(* IEC 61131-3 sources: ST_DesignPattern/Behavioral, 4 files *)

(* ---- adapter.st ---- *)
{attribute 'qualified_only'}
{attribute 'strict'}
{attribute 'to_string'}
TYPE E_GasSystemType:
(
    PRECURSOR := 0,
    REACTANT := 1,
    INERT := 2
);
END_TYPE

{attribute 'qualified_only'}
{attribute 'strict'}
{attribute 'to_string'}
TYPE E_MFCState:
(
    Idle := 0,
    Running := 10,
    Error := 20
);
END_TYPE

TYPE ST_MFCConfig :
STRUCT
    fMaxFlow    : REAL;
    fMinFlow    : REAL;
    fTolerance  : REAL;
    sName       : STRING;
    sFlowUnit   : STRING := 'sccm';
END_STRUCT
END_TYPE

INTERFACE I_MFC
    METHOD SetFlow : BOOL
    VAR_INPUT
        fSetpoint : REAL;
    END_VAR
    END_METHOD

    METHOD GetFlow : REAL
    END_METHOD

    METHOD AtSetpoint : BOOL
    END_METHOD

    METHOD Stop : BOOL
    END_METHOD

    PROPERTY State : E_MFCState GET
    END_PROPERTY

    PROPERTY Error : ST_Error GET
    END_PROPERTY
END_INTERFACE

FUNCTION_BLOCK FB_MFC IMPLEMENTS I_MFC
VAR
    _config : ST_MFCConfig;
    _state : E_MFCState := E_MFCState.Idle;
    _errorHandler : FB_ErrorHandler;
    _pMFC : POINTER TO massFlowController;
END_VAR

VAR CONSTANT
    ZERO_FLOW_THRESHOLD : REAL := 0.001;
END_VAR

METHOD Initialize : BOOL
VAR_INPUT
    config: ST_MFCConfig;
    pMFC: POINTER TO massFlowController;
END_VAR
    _config := config;
    _pMFC := pMFC;
    _errorHandler := errorHandler;

    IF _pMFC = 0 THEN
        _errorHandler.RegisterError(
            eErrorCode := E_ErrorCodes.NotInitialized,
            eCategory := E_ErrorCategory.Hardware,
            sComponent := _config.sName,
            sDescription := 'MFC hardware not connected',
            sCurrentValue := '',
            sExpectedValue := '',
            sUnit := ''
        );
        _state := E_MFCState.Error;
        Initialize := FALSE;
        RETURN;
    END_IF

    Initialize := TRUE;
END_METHOD

METHOD SetFlow : BOOL
VAR_INPUT
    fSetpoint : REAL;
END_VAR
    IF _pMFC = 0 THEN
        _errorHandler.RegisterError(
            eErrorCode := E_ErrorCodes.NotInitialized,
            eCategory := E_ErrorCategory.Hardware,
            sComponent := _config.sName,
            sDescription := 'MFC hardware not connected',
            sCurrentValue := '',
            sExpectedValue := '',
            sUnit := ''
        );
        _state := E_MFCState.Error;
        SetFlow := FALSE;
        RETURN;
    END_IF

    IF fSetpoint < _config.fMinFlow OR fSetpoint > _config.fMaxFlow THEN
        _errorHandler.RegisterError(
            eErrorCode := E_ErrorCodes.FlowOutOfRange,
            eCategory := E_ErrorCategory.FlowControl,
            sComponent := _config.sName,
            sDescription := 'Flow setpoint out of range',
            sCurrentValue := REAL_TO_STRING(fSetpoint),
            sExpectedValue := CONCAT(LREAL_TO_STRING(_config.fMinFlow), CONCAT(' - ', LREAL_TO_STRING(_config.fMaxFlow))),
            sUnit := 'sccm'
        );
        _state := E_MFCState.Error;
        RETURN;
    END_IF

    _pMFC^.SetPointIn := fSetpoint;
    _state := SEL(fSetpoint = 0, E_MFCState.Running, E_MFCState.Idle);
    SetFlow := TRUE;
END_METHOD

METHOD GetFlow : REAL
    IF _pMFC <> 0 THEN
        GetFlow := _pMFC^.ProcessValue;
    END_IF
END_METHOD

METHOD AtSetpoint : BOOL
    IF _pMFC = 0 THEN
        AtSetpoint := FALSE;
        RETURN;
    END_IF

    AtSetpoint := ABS(_pMFC^.ProcessValue - _pMFC^.SetPointIn) <= (_pMFC^.SetPointIn * _config.fTolerance / 100.0);
END_METHOD

METHOD Stop : BOOL
    Stop := SetFlow(0.0);
END_METHOD

PROPERTY State : E_MFCState GET
    State := _state;
END_PROPERTY

PROPERTY Error : ST_Error GET
    Error := _errorHandler.GetError();
END_PROPERTY
END_FUNCTION_BLOCK

FUNCTION_BLOCK FB_DualMFC IMPLEMENTS I_MFC
VAR
    _highFlow: FB_MFC;
    _lowFlow: FB_MFC;
    _flowThreshold: REAL;
    _activeFlow: REFERENCE TO FB_MFC;
    _state: E_MFCState := E_MFCState.Idle;
    _errorHandler: FB_ErrorHandler;
END_VAR

METHOD Initialize : BOOL
VAR_INPUT
    highConfig: ST_MFCConfig;
    lowConfig: ST_MFCConfig;
    pHighMFC: POINTER TO massFlowController;
    pLowMFC: POINTER TO massFlowController;
    errorHandler: I_ErrorHandler;
END_VAR
    _errorHandler := errorHandler;

    IF NOT _highFlow.Initialize(highConfig, pHighMFC, _errorHandler) THEN
        _errorHandler.RegisterError(
            eErrorCode := E_ErrorCodes.MFCTimeout,
            eCategory := E_ErrorCategory.Initialization,
            sComponent := 'DualMFC-High',
            sDescription := 'Failed to initialize high flow MFC',
            sCurrentValue := '',
            sExpectedValue := '',
            sUnit := ''
        );
        _state := E_MFCState.Error;
        RETURN FALSE;
    END_IF

    IF NOT _lowFlow.Initialize(lowConfig, pLowMFC, _errorHandler) THEN
        _errorHandler.RegisterError(
            eErrorCode := E_ErrorCodes.MFCTimeout,
            eCategory := E_ErrorCategory.Initialization,
            sComponent := 'DualMFC-Low',
            sDescription := 'Failed to initialize low flow MFC',
            sCurrentValue := '',
            sExpectedValue := '',
            sUnit := ''
        );
        _state := E_MFCState.Error;
        RETURN FALSE;
    END_IF

    _flowThreshold := lowConfig.fMaxFlow;
    _activeFlow REF= _lowFlow;
    _state := E_MFCState.Idle;
    Initialize := TRUE;
END_METHOD

METHOD SetFlow : BOOL
VAR_INPUT
    fSetpoint : REAL;
END_VAR
    IF _state = E_MFCState.Error THEN
        RETURN FALSE;
    END_IF

    IF fSetpoint <= _flowThreshold THEN
        _highFlow.Stop();
        _activeFlow REF= _lowFlow;
    ELSE
        _lowFlow.Stop();
        _activeFlow REF= _highFlow;
    END_IF

    SetFlow := _activeFlow.SetFlow(fSetpoint);
    _state := _activeFlow.State;
END_METHOD

METHOD GetFlow : REAL
    GetFlow := _lowFlow.GetFlow() + _highFlow.GetFlow();
END_METHOD

METHOD Stop : BOOL
    _highFlow.Stop();
    _lowFlow.Stop();
    _state := E_MFCState.Idle;
    Stop := TRUE;
END_METHOD

METHOD AtSetpoint : BOOL
    IF _state = E_MFCState.Error THEN
        RETURN FALSE;
    END_IF

    AtSetpoint := _activeFlow.AtSetpoint();
END_METHOD

PROPERTY State : E_MFCState GET
    State := _state;
END_PROPERTY

PROPERTY Error : ST_Error GET
    IF _activeFlow.State = E_MFCState.Error THEN
        Error := _activeFlow.Error;
    ELSE
        Error := _errorHandler.GetError();
    END_IF
END_PROPERTY
END_FUNCTION_BLOCK

FUNCTION_BLOCK FB_MFCFactory
VAR CONSTANT
    PRECURSOR_HIGH_CONFIG : ST_MFCConfig := (
        fMaxFlow := 2000.0,
        fMinFlow := 400.0,
        fTolerance := 2.0,
        sName := 'Precursor High Flow',
        sFlowUnit := 'sccm'
    );

    PRECURSOR_LOW_CONFIG : ST_MFCConfig := (
        fMaxFlow := 400.0,
        fMinFlow := 0.0,
        fTolerance := 2.0,
        sName := 'Precursor Low Flow',
        sFlowUnit := 'sccm'
    );

    REACTANT_CONFIG : ST_MFCConfig := (
        fMaxFlow := 1000.0,
        fMinFlow := 0.0,
        fTolerance := 2.0,
        sName := 'Reactant Flow',
        sFlowUnit := 'sccm'
    );

    INERT_HIGH_CONFIG : ST_MFCConfig := (
        fMaxFlow := 5000.0,
        fMinFlow := 400.0,
        fTolerance := 2.0,
        sName := 'Inert High Flow',
        sFlowUnit := 'sccm'
    );

    INERT_LOW_CONFIG : ST_MFCConfig := (
        fMaxFlow := 400.0,
        fMinFlow := 0.0,
        fTolerance := 2.0,
        sName := 'Inert Low Flow',
        sFlowUnit := 'sccm'
    );
END_VAR

VAR
    _reactantMFC : FB_MFC;
    _precursorDualMFC : FB_DualMFC;
    _inertDualMFC : FB_DualMFC;
    _errorHandler : I_ErrorHandler;
    _bInitialized : BOOL := FALSE;

END_VAR

METHOD Initialize : BOOL
VAR_INPUT
    bResetError : BOOL := FALSE;
    errorHandler : I_ErrorHandler;
END_VAR
    _errorHandler := errorHandler;

    IF bResetError THEN
        _errorHandler.Reset();
    END_IF

    IF _bInitialized THEN
        Initialize := TRUE;
        RETURN;
    END_IF

    IF NOT _reactantMFC.Initialize(REACTANT_CONFIG, ADR(GVL_E02_MFC.MFC.st_MFC.ReactantMassFlowController1), _errorHandler) THEN
        _errorHandler.RegisterError(
            eErrorCode := E_ErrorCodes.MFCTimeout,
            eCategory := E_ErrorCategory.Initialization,
            sComponent := REACTANT_CONFIG.sName,
            sDescription := 'Failed to initialize reactant MFC',
            sCurrentValue := '',
            sExpectedValue := '',
            sUnit := REACTANT_CONFIG.sFlowUnit
        );
        RETURN;
    END_IF

    IF NOT _precursorDualMFC.Initialize(PRECURSOR_HIGH_CONFIG, PRECURSOR_LOW_CONFIG, ADR(GVL_E02_MFC.MFC.st_MFC.PrecursorMassFlowController1), ADR(GVL_E02_MFC.MFC.st_MFC.PrecursorMassFlowController2), _errorHandler) THEN
        _errorHandler.RegisterError(
            eErrorCode := E_ErrorCodes.MFCTimeout,
            eCategory := E_ErrorCategory.Initialization,
            sComponent := 'Precursor Dual MFC',
            sDescription := 'Failed to initialize precursor dual MFC',
            sCurrentValue := '',
            sExpectedValue := '',
            sUnit := PRECURSOR_HIGH_CONFIG.sFlowUnit
        );
        RETURN;
    END_IF

    IF NOT _inertDualMFC.Initialize(INERT_HIGH_CONFIG, INERT_LOW_CONFIG, ADR(GVL_E02_MFC.MFC.st_MFC.InertMassFlowController1), ADR(GVL_E02_MFC.MFC.st_MFC.InertMassFlowController2), _errorHandler) THEN
        _errorHandler.RegisterError(
            eErrorCode := E_ErrorCodes.MFCTimeout,
            eCategory := E_ErrorCategory.Initialization,
            sComponent := 'Inert Dual MFC',
            sDescription := 'Failed to initialize inert dual MFC',
            sCurrentValue := '',
            sExpectedValue := '',
            sUnit := INERT_HIGH_CONFIG.sFlowUnit
        );
        RETURN;
    END_IF

    _bInitialized := TRUE;
    Initialize := TRUE;
END_METHOD

METHOD GetController : REFERENCE TO I_MFC
VAR_INPUT
    eGasType : E_GasSystemType;
END_VAR
    IF NOT _bInitialized THEN
        _errorHandler.RegisterError(
            eErrorCode := E_ErrorCodes.NotInitialized,
            eCategory := E_ErrorCategory.Initialization,
            sComponent := 'MFCFactory',
            sDescription := 'Factory not initialized',
            sCurrentValue := '',
            sExpectedValue := '',
            sUnit := ''
        );
        RETURN;
    END_IF

    CASE eGasType OF
        E_GasSystemType.PRECURSOR:
            GetController REF= _precursorDualMFC;

        E_GasSystemType.REACTANT:
            GetController REF= _reactantMFC;

        E_GasSystemType.INERT:
            GetController REF= _inertDualMFC;

        ELSE
            _errorHandler.RegisterError(
                eErrorCode := E_ErrorCodes.InvalidConfiguration,
                eCategory := E_ErrorCategory.FlowControl,
                sComponent := 'MFCFactory',
                sDescription := 'Invalid gas system type',
                sCurrentValue := TO_STRING(eGasType),
                sExpectedValue := 'PRECURSOR, REACTANT, or INERT',
                sUnit := ''
            );
    END_CASE
END_METHOD

PROPERTY Error : ST_Error GET
    Error := _errorHandler.GetError();
END_PROPERTY
END_FUNCTION_BLOCK

(* ---- bridge.st ---- *)
FUNCTION_BLOCK ABSTRACT FB_Shape
VAR
	_color : ITF_color;
END_VAR
    METHOD FB_init : BOOL
    VAR_INPUT
        bInitRetains : BOOL; // if TRUE, the retain variables are initialized (warm start / cold start)
        bInCopyCode : BOOL;  // if TRUE, the instance afterwards gets moved into the copy code (online change)
        Color : ITF_Color;
    END_VAR
        THIS^._color := Color;
    END_METHOD

    METHOD ABSTRACT Draw : STRING
    END_METHOD
END_FUNCTION_BLOCK

FUNCTION_BLOCK FB_Square EXTENDS FB_Shape
    METHOD Draw : STRING
        ADSLOGSTR(    msgCtrlMask:=ADSLOG_MSGTYPE_LOG,
              msgFmtStr:='Drawing a %s square',
              strArg:= SUPER^._color.applyColor());
    END_METHOD
END_FUNCTION_BLOCK

FUNCTION_BLOCK FB_Circle EXTENDS FB_Shape
    METHOD Draw : STRING
        ADSLOGSTR(    msgCtrlMask:=ADSLOG_MSGTYPE_LOG,
              msgFmtStr:='Drawing a %s circle',
              strArg:= SUPER^._color.applyColor());
    END_METHOD
END_FUNCTION_BLOCK

INTERFACE ITF_Color
    METHOD applyColor : STRING
    END_METHOD
END_INTERFACE

FUNCTION_BLOCK FB_BlueColor IMPLEMENTS ITF_Color
    METHOD applyColor : STRING
        applyColor := 'blue';
    END_METHOD
END_FUNCTION_BLOCK

FUNCTION_BLOCK FB_RedColor IMPLEMENTS ITF_Color
    METHOD applyColor : STRING
        applyColor := 'red';
    END_METHOD
END_FUNCTION_BLOCK

PROGRAM MAIN
VAR

     fbRedColor 		: FB_RedColor;
	 fbBlueColor 		: FB_BlueColor;

	 fbSquareRed 		: FB_Square(Color:= fbRedColor );
	 fbSquareBlue 		: FB_Square(Color:= fbBlueColor );

	 fbCircleRed 		: FB_Circle(Color:= fbRedColor );
	 fbCircleBlue 		: FB_Circle(Color:= fbBlueColor );

	 bstartDemo1		: BOOL;

END_VAR
    IF bstartDemo1 THEN
        bstartDemo1 := FALSE;

        fbSquareRed.Draw();
        fbSquareBlue.Draw();

        fbCircleRed.Draw();
        fbCircleBlue.Draw();

    END_IF
END_PROGRAM

(* ---- composite.st ---- *)
INTERFACE I_Component
    METHOD AddChild
    VAR_INPUT
        Child : I_Component;
    END_VAR
    END_METHOD

    METHOD GetChildren : ARRAY [1..Param.NumberOfChildren] OF I_Component;
    END_METHOD

    PROPERTY GetSize : INT GET
    END_PROPERTY
END_INTERFACE

FUNCTION_BLOCK ABSTRACT Component IMPLEMENTS I_component
VAR
	_name : STRING;
END_VAR
    METHOD FB_init : BOOL
    VAR_INPUT
        bInitRetains : BOOL; // if TRUE, the retain variables are initialized (warm start / cold start)
        bInCopyCode : BOOL;  // if TRUE, the instance afterwards gets moved into the copy code (online change)
        name : STRING;
    END_VAR
    THIS^._name := name;
    END_METHOD

    METHOD ABSTRACT AddChild
    VAR_INPUT
        Child : I_Component;
    END_VAR
    END_METHOD

    METHOD ABSTRACT GetChildren : ARRAY [1..Param.NumberOfChildren] OF I_Component;
    END_METHOD

    PROPERTY ABSTRACT GetSize : INT GET
    END_PROPERTY

    PROPERTY Name : STRING GET
        Name := THIS^._name;
    END_PROPERTY
END_FUNCTION_BLOCK

FUNCTION_BLOCK Archive EXTENDS Component
VAR
//	_name : STRING;
	_size : INT;
END_VAR
    METHOD FB_init : BOOL
    VAR_INPUT
        bInitRetains : BOOL; // if TRUE, the retain variables are initialized (warm start / cold start)
        bInCopyCode : BOOL;  // if TRUE, the instance afterwards gets moved into the copy code (online change)
        name : STRING;
        iSize : INT;
    END_VAR
        THIS^._name := name;
        THIS^._size := iSize
    END_METHOD

    METHOD AddChild
    VAR_INPUT
        Child : I_Component;
    END_VAR
    END_METHOD

    METHOD GetChildren : ARRAY [1..Param.NumberOfChildren] OF I_Component;
    VAR_INPUT
    END_VAR
    END_METHOD

    PROPERTY GetSize : INT GET
        GetSize := _size;
    END_PROPERTY
END_FUNCTION_BLOCK

FUNCTION_BLOCK Directory EXTENDS Component
VAR
	children 			: ARRAY [1..Param.NumberOfChildren] OF I_Component;
	childCount			: INT := 0;
END_VAR
    METHOD AddChild
    VAR_INPUT
        Child : I_Component;
    END_VAR
    VAR
        i: INT;
    END_VAR
        childCount := childCount + 1;
        children[childCount] := Child;
    END_METHOD

    METHOD GetChildren : ARRAY [1..Param.NumberOfChildren] OF I_Component;
        GetChildren := children;
    END_METHOD

    PROPERTY GetSize : INT
    VAR
        i : INT := 0;
    END_VAR
        FOR i := 1 TO childCount  DO
            GetSize := GetSize + children[i].GetSize;
        END_FOR
    END_PROPERTY

    METHOD ResetSize
        childCount:= 0;
    END_METHOD
END_FUNCTION_BLOCK

PROGRAM MAIN
VAR
	root 		: Directory('root');

	archive1	: Archive('archivo1.txt', 10);
    archive2  	: Archive('archivo2.txt', 30);
    archive3 	: Archive('archivo3.txt', 120);
    archive4 	: Archive('archivo4.txt', 800);
    archive5 	: Archive('archivo5.txt', 340);

    archive6 	: Archive('archivo6.txt', 122);
    archive7 	: Archive('archivo7.txt', 391);

    dir1 		: Directory('dir1');
    dir2 		: Directory('dir2');
    dir3 		: Directory('dir3');

	bExecute	: BOOL;
	sMsg 		: STRING;
END_VAR
    IF bExecute THEN

        bExecute := FALSE;

        dir1.ResetSize();
        dir2.ResetSize();
        dir3.ResetSize();
        root.ResetSize();

        dir1.AddChild(archive1); // 10
        dir1.AddChild(archive6); // 122
        dir2.AddChild(archive2); // 30
        dir3.AddChild(archive3); // 120
        dir3.AddChild(archive4); // 800
        dir1.AddChild(dir3); // 120+800

        root.AddChild(dir1); // dir1 = 120+800+10+122 = 1052
        root.AddChild(dir2); // dir2 = 30
        root.AddChild(archive5); // 340
        root.AddChild(archive7); // 391

        // root = 1052+30+340+391 = 1813
        sMsg := CONCAT(STR1:= root.Name , STR2:= CONCAT(STR1:= ' is: ' , STR2:= TO_STRING(root.GetSize) ) );
        ADSLOGSTR(msgCtrlMask:= ADSLOG_MSGTYPE_LOG, msgFmtStr:= 'The size of the directory %s ' , strArg:= sMsg);

        // dir1 = 10+122+120+800 = 1052
        sMsg := CONCAT(STR1:= dir1.Name , STR2:= CONCAT(STR1:= ' is: ' , STR2:= TO_STRING(dir1.GetSize) ) );
        ADSLOGSTR(msgCtrlMask:= ADSLOG_MSGTYPE_LOG, msgFmtStr:= 'The size of the directory %s ' , strArg:= sMsg);

        // dir2 = 30
        sMsg := CONCAT(STR1:= dir2.Name , STR2:= CONCAT(STR1:= ' is: ' , STR2:= TO_STRING(dir2.GetSize) ) );
        ADSLOGSTR(msgCtrlMask:= ADSLOG_MSGTYPE_LOG, msgFmtStr:= 'The size of the directory %s ' , strArg:= sMsg);

        // dir3 = 120+800 = 922
        sMsg := CONCAT(STR1:= dir3.Name , STR2:= CONCAT(STR1:= ' is: ' , STR2:= TO_STRING(dir3.GetSize) ) );
        ADSLOGSTR(msgCtrlMask:= ADSLOG_MSGTYPE_LOG, msgFmtStr:= 'The size of the directory %s ' , strArg:= sMsg);
    END_IF
END_PROGRAM

(* ---- decorator.st ---- *)
INTERFACE I_Shape
    METHOD M_Draw: BOOL
    END_METHOD
END_INTERFACE

FUNCTION_BLOCK FB_Circle IMPLEMENTS I_Shape
    METHOD M_Draw: BOOL
        ADSLOGSTR(ADSLOG_MSGTYPE_HINT, 'Draw circle', '');
        M_Draw := TRUE;
    END_METHOD
END_FUNCTION_BLOCK

FUNCTION_BLOCK FB_Square IMPLEMENTS I_Shape
    METHOD M_Draw: BOOL
        ADSLOGSTR(ADSLOG_MSGTYPE_HINT, 'Draw Square', '');
        M_Draw := TRUE;
    END_METHOD
END_FUNCTION_BLOCK

FUNCTION_BLOCK ABSTRACT FB_ShapeDecorator IMPLEMENTS I_Shape
VAR
	_iDecoratedShape: I_Shape;
END_VAR
    METHOD FB_init: BOOL
    VAR_INPUT
        bInitRetains: BOOL; // if TRUE, the retain variables are initialized (warm start / cold start)
        bInCopyCode: BOOL; // if TRUE, the instance afterwards gets moved into the copy code (online change)
        iDecoratedShape: I_Shape;
    END_VAR
        _iDecoratedShape := iDecoratedShape;
    END_METHOD

    METHOD ABSTRACT M_Draw: BOOL
    END_METHOD
END_FUNCTION_BLOCK

{attribute 'qualified_only'}
{attribute 'strict'}
TYPE E_BorderDashType:
(
	Solid := 0,
	RoundDot,
	SquareDot,
	Dash,
	LongDashDot
);
END_TYPE

FUNCTION_BLOCK FB_BorderDashTypeDecorator EXTENDS FB_ShapeDecorator
VAR
	_eBorderDashType: E_BorderDashType;
END_VAR
    METHOD FB_init: BOOL
    VAR_INPUT
        bInitRetains: BOOL; // if TRUE, the retain variables are initialized (warm start / cold start)
        bInCopyCode: BOOL; // if TRUE, the instance afterwards gets moved into the copy code (online change)
        iDecoratedShape: I_Shape;
        eBorderDashType: E_BorderDashType;
    END_VAR
        SUPER^._iDecoratedShape := iDecoratedShape;
        _eBorderDashType := eBorderDashType;
    END_METHOD

    METHOD M_Draw: BOOL
        M_Draw := SUPER^._iDecoratedShape.M_Draw();
        M_SetBorderDashType(SUPER^._iDecoratedShape);
    END_METHOD

    METHOD M_SetBorderDashType
    VAR_INPUT
        iDecoratedShape: I_Shape;
    END_VAR
        CASE _eBorderDashType OF
            E_BorderDashType.Solid:
                ADSLOGSTR(ADSLOG_MSGTYPE_HINT, 'Border Dash Type: Solid', '');

            E_BorderDashType.SquareDot:
                ADSLOGSTR(ADSLOG_MSGTYPE_HINT, 'Border Dash Type: Square Dot', '');

            E_BorderDashType.RoundDot:
                ADSLOGSTR(ADSLOG_MSGTYPE_HINT, 'Border Dash Type: Round Dot', '');

            E_BorderDashType.Dash:
                ADSLOGSTR(ADSLOG_MSGTYPE_HINT, 'Border Dash Type: Dash', '');

            E_BorderDashType.LongDashDot:
                ADSLOGSTR(ADSLOG_MSGTYPE_HINT, 'Border Dash Type:Long Dash Dot', '');

        ELSE
            ADSLOGSTR(ADSLOG_MSGTYPE_HINT, 'Border Dash Type:Unkown', '');
        END_CASE
    END_METHOD

    PROPERTY P_GS_BorderDashType: E_BorderDashType
        GET:
            P_GS_BorderDashType := _eBorderDashType;
        SET:
            _eBorderDashType := P_GS_BorderDashType;
    END_PROPERTY
END_FUNCTION_BLOCK

FUNCTION_BLOCK FB_GreenShapeDecorator EXTENDS FB_ShapeDecorator
    METHOD FB_init: BOOL
    VAR_INPUT
        bInitRetains: BOOL; // if TRUE, the retain variables are initialized (warm start / cold start)
        bInCopyCode: BOOL; // if TRUE, the instance afterwards gets moved into the copy code (online change)
        iDecoratedShape: I_Shape;
    END_VAR
        SUPER^._iDecoratedShape := iDecoratedShape;
    END_METHOD

    METHOD M_Draw: BOOL
        M_Draw := SUPER^._iDecoratedShape.M_Draw();
        M_SetGreenBorder(SUPER^._iDecoratedShape);
    END_METHOD

    METHOD PRIVATE M_SetGreenBorder
    VAR_INPUT
        iDecoratedShape: I_Shape;
    END_VAR
        ADSLOGSTR(ADSLOG_MSGTYPE_HINT, 'Border Color: Green', '');
    END_METHOD
END_FUNCTION_BLOCK

PROGRAM MAIN
VAR
	fbCircle: FB_Circle;
	fbGreenCircle: FB_GreenShapeDecorator(fbCircle);
	fbRoundDotBorderGreenCircle: FB_BorderDashTypeDecorator(fbGreenCircle, E_BorderDashType.RoundDot);

	fbSquare: FB_Square;
	fbGreenSquare: FB_GreenShapeDecorator(fbSquare);
	fbDashBorderGreenSquare: FB_BorderDashTypeDecorator(fbGreenSquare, E_BorderDashType.Dash);

	bDemoStart: BOOL;
END_VAR
    IF bDemoStart THEN

        bDemoStart := FALSE;

        fbRoundDotBorderGreenCircle.M_Draw();

        fbDashBorderGreenSquare.M_Draw();

    END_IF
END_PROGRAM
